RoboDK station: Ruta_DER.rdk

Station Ruta_DER (saved by RoboDK 5.5.4). Poses are relative to the parent item; angles as X-Y-Z fixed-axis rotations.
  - object R7 at (0, 0, 0) mm
